FUNCTION_BLOCK ABSTRACT T_NullableBaseClass
VAR
	_Stubbed : BOOL;
END_VAR

METHOD Stub
VAR_INPUT

END_VAR
_Stubbed := TRUE;
END_METHOD

PROPERTY Stubbed : BOOL
GET
Stubbed := _Stubbed;
END_GET
END_PROPERTY

END_FUNCTION_BLOCK

(* stored: Version 1.1.0.1, ProductVersion 3.1.4024.12
   POU T_NullableBaseClass: Id {6918528b-1f2d-49da-b5a1-1e8c3d318bfe}, SpecialFunc None
   Method Stub: Id {d096dc91-6a78-4247-b9c0-a385b806bf7a}
   Property Stubbed: Id {5b0c7159-d46a-4902-aa32-4a6d5b18f358}
   Get Get: Id {2aa51fea-b957-4959-890e-4dedfdacb9e4} *)
